Omron Sysmac Studio project modbus_tcp_server (Sysmac Studio 1.47.0.64008, StandardProject)

# Controller new_Controller_0: NX1P2-9024DT version 1.40
Task PrimaryTask (priority 4, period or condition 2000): Program0
Library OEN_Communication_V1_0_22 1.0.22 (contents left out)

PROGRAM Program0
VAR
    T1000ms : TIME;
    T100ms : TIME;
    mod_request : ARRAY[0..2] OF OEN\Modbus\sModbusReq := [(Enable := True, NodeAdr := 0, FunctionCode := Fn03_ReadHoldingRegisters, Read := (StartAddressRemote := 0, StartAddressLocal := 0, Count := 3), Write := (StartAddressRemote := 0, StartAddressLocal := 0, Count := 0)), (Enable := True, NodeAdr := 0, FunctionCode := Fn16_WriteMultipleRegisters, Read := (StartAddressRemote := 0, StartAddressLocal := 0, Count := 0), Write := (StartAddressRemote := 3, StartAddressLocal := 3, Count := 3)), (Enable := True, NodeAdr := 0, FunctionCode := Fn04_ReadInputRegisters, Read := (StartAddressRemote := 7, StartAddressLocal := 7, Count := 4), Write := (StartAddressRemote := 0, StartAddressLocal := 0, Count := 0))];
    mod_coils : ARRAY[0..10] OF BOOL;
    mod_discre_input : ARRAY[0..10] OF BOOL;
    mod_input_register : ARRAY[0..10] OF WORD;
    Holding_register : ARRAY[0..10] OF WORD;
    functio_modbus_client : OEN\Modbus\ModbusTCP_Client;
END_VAR

(* Section Section0: ladder, written here as Structured Text *)

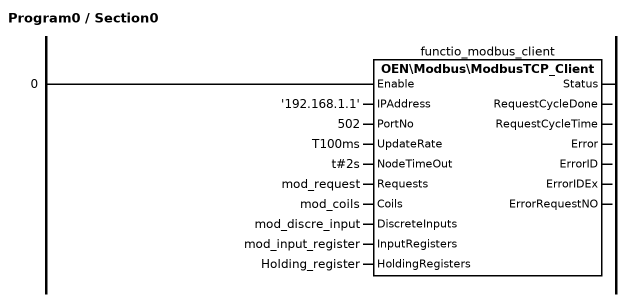
(* Rung 0 *)
functio_modbus_client(Enable := TRUE, IPAddress := '192.168.1.1', PortNo := 502, UpdateRate := T100ms, NodeTimeOut := t#2s, Requests := mod_request, Coils := mod_coils, DiscreteInputs := mod_discre_input, InputRegisters := mod_input_register, HoldingRegisters := Holding_register);
END_PROGRAM